{attribute addProperty BoxType "EP2339-0042-0017"}
{attribute addProperty Id "OutputAT %Q*BOOL81"}
{attribute addProperty CRC "2134331056"}
{attribute addProperty SizeInBites "8"}
{attribute addProperty SizeInBytes "1"}
TYPE DO_X04_Pin_7F374EB0 :
STRUCT
	{attribute addProperty Name "Output"}
	Output AT %Q* : BOOL;
END_STRUCT
END_TYPE

(* stored: Version 1.2.0.0, ProductVersion 3.1.4024.9
   DUT DO_X04_Pin_7F374EB0: Id {5a4202bf-2a4c-4d9d-abcd-482535bb78cd} *)
